// TIA Portal V19 export
VAR_GLOBAL   // PLC tag table "LB322"
   LB322_AssiemaggioBordatura_Pb_Aux2 AT %I252.2 : Bool;   // 355SH2
   LB322_AssiemaggioBordatura_Pb_Aux1 AT %I252.1 : Bool;   // 355SH1
   LB322_AssiemaggioBordatura_Lp_Aux2 AT %Q251.6 : Bool;   // 355SH2
   LB322_AssiemaggioBordatura_Lp_Aux1 AT %Q251.5 : Bool;   // 355SH1
END_VAR
